Fanuc KAREL source: kt00267.KL

-- PROVISIONAL review KL for V770-1; original PC SHA256 7dbe4daf749bda1d6ec26f5e132bd2c9a89f9005e438596d34a2ddda012b672f
-- Incomplete behavior may be omitted. Consult companion uncertainty JSON. Do not deploy.
PROGRAM KT00267
%NOLOCKGROUP
VAR
  I2 : INTEGER
  OUT : BOOLEAN
-- UNRESOLVED_DECL Y1 type=002018
BEGIN
  -- UNRESOLVED_PC offsets 5-19; opcodes 2E,22,9D,33,B2
  -- UNRESOLVED_PC offsets 24-35; opcodes 2E,23
  -- UNRESOLVED_PC offsets 40-62; opcodes 22,9D,33,B1,21,57,23
  -- UNRESOLVED_PC offsets 67-71; opcodes 7F
END KT00267
